TYPE csp_case_tr_accU_virtualMaster_enum :
(
	CSP_CASE_TR_ACCU_VIRTUAL_MASTER_STATUS_NOT_INITIALIZED 								:= 0,
	CSP_CASE_TR_ACCU_VIRTUAL_MASTER_STATUS_DISABLED 									:= 10,
	CSP_CASE_TR_ACCU_VIRTUAL_MASTER_STATUS_POSITION_CHECK								:= 20,
	CSP_CASE_TR_ACCU_VIRTUAL_MASTER_STATUS_CHECK_SLAVE_GEAR 							:= 25,
	CSP_CASE_TR_ACCU_VIRTUAL_MASTER_STATUS_ENABLE_REQUEST 								:= 30,
	CSP_CASE_TR_ACCU_VIRTUAL_MASTER_STATUS_ENABLED 										:= 40,
	CSP_CASE_TR_ACCU_VIRTUAL_MASTER_STATUS_ABS_MOVE_REQUEST								:= 50,
	CSP_CASE_TR_ACCU_VIRTUAL_MASTER_STATUS_ABS_MOVING									:= 60,
	CSP_CASE_TR_ACCU_VIRTUAL_MASTER_STATUS_STOP_REQUEST 								:= 70,
	CSP_CASE_TR_ACCU_VIRTUAL_MASTER_STATUS_DISABLE_REQUEST 								:= 80,
	CSP_CASE_TR_ACCU_VIRTUAL_MASTER_STATUS_DISABLING 									:= 90
) := CSP_CASE_TR_ACCU_VIRTUAL_MASTER_STATUS_NOT_INITIALIZED;
END_TYPE

(* stored: Version 1.1.0.1, ProductVersion 3.1.4024.3
   DUT csp_case_tr_accU_virtualMaster_enum: Id {c5ba65bf-a49d-4d3f-9037-0b2b595e6651} *)
